FUNCTION_BLOCK FB_YokeInputScaling
VAR_INPUT
	bEnable 				: BOOL;
	nRawInput 				: INT;
	stYokeInputScaling  	: ST_YokeInputScaling;
END_VAR
VAR_OUTPUT
	fNormalizedOutput 		: LREAL;
END_VAR
VAR
	fRawInput 				: LREAL;
	fTempInput 				: LREAL;
	fTempOutput 			: LREAL;
END_VAR

fRawInput := INT_TO_LREAL(nRawInput);

fTempInput := fRawInput - stYokeInputScaling.fNeutralInputValue;

IF fTempInput > stYokeInputScaling.fNeutralDeadband THEN
	fTempOutput := fTempInput/(stYokeInputScaling.fMaxInputValue - stYokeInputScaling.fNeutralInputValue);
ELSIF fTempInput < -stYokeInputScaling.fNeutralDeadband THEN	
	fTempOutput := fTempInput/(stYokeInputScaling.fNeutralInputValue - stYokeInputScaling.fMinInputValue);
ELSE
	fTempOutput := 0.0;
END_IF

IF NOT(bEnable) THEN
	fNormalizedOutput := 0.0;
ELSE
	fNormalizedOutput := LIMIT(stYokeInputScaling.fMinOutputValue, fTempOutput, stYokeInputScaling.fMaxOutputValue); 
END_IF

END_FUNCTION_BLOCK

(* stored: Version 1.1.0.1, ProductVersion 3.1.4026.11
   POU FB_YokeInputScaling: Id {7ea0edf3-703a-4e77-8eb7-84184ece0335}, SpecialFunc None *)
